// TIA Portal V20 export
DATA_BLOCK "IDB_GlobalStatus"   // DB48
// stored: InstanceOfName Global.FB_GlobalStatus, InstanceOfType FB, Namespace Global
"Global.FB_GlobalStatus"
   // VAR
   //    Line : Struct
   //       ProductionLine : "Global.ConveyorStatus";
   //       EmptyLine { S7_SetPoint := 'True'} : "Global.ConveyorStatus";
   //       PackedLine { S7_SetPoint := 'True'} : "Global.ConveyorStatus";
   //    END_STRUCT;
   //    cmp : Struct
   //       ProductionTotes_Value0 : Array[_.gminProductionLine.._.gmaxProductionLine] of Bool;
   //       ProductionTotes_Value1 : Array[_.gminProductionLine.._.gmaxProductionLine] of Bool;
   //       EmptyLine_Value0 : Array[_.gminEmptyLine.._.gmaxEmptyLine] of Bool;
   //       EmptyLine_Value1 : Array[_.gminEmptyLine.._.gmaxEmptyLine] of Bool;
   //       PackedLine_Value0 : Array[_.gminPackedLine.._.gmaxPackedLine] of Bool;
   //       PackedLine_Value1 : Array[_.gminPackedLine.._.gmaxPackedLine] of Bool;
   //    END_STRUCT;
   //    ForVisu : Struct
   //       Line : Struct
   //          ProductionLine : Word;
   //          EmptyLine : Word;
   //          PackedLine : Word;
   //       END_STRUCT;
   //    END_STRUCT;
   // END_VAR
BEGIN
   cmp.ProductionTotes_Value1[1001..1192] := True;
   cmp.EmptyLine_Value1[2001..2109] := True;
   cmp.PackedLine_Value1[3001..3040] := True;
END_DATA_BLOCK
